FUNCTION_BLOCK TmsHoldStation EXTENDS Process 
VAR
	_EmbarkStation : IStation;
	ExecuteSeqeunce : BOOL;
	HoldMover : I_XtsMover;
	State :(
		Init,                                               
		Ready,                                 
        Waiting,
		Processing,
		Clearing,
		Aborting); 
END_VAR

{analysis -2}

METHOD PUBLIC  Cycle : HRESULT
VAR
	CycleResult : HRESULT;
END_VAR
Cycle := S_OK;
CASE State OF
	Init:
		_Operating := _IsClear := _Complete := _Ready := _HasMover := FALSE;
		StationMovers := 0;
		State := Ready;
	
	Ready:	
		IF ExecuteSeqeunce THEN
			_Operating := _Complete := _HasMover := FALSE;
			_IsClear := _Ready := TRUE;
			StationMovers := 0;
			State := Waiting;
		END_IF
	
	Waiting:
		IF _HasMover THEN
			State := Processing;
			_Operating := TRUE;
			_IsClear := FALSE;
			_Ready := FALSE;
		END_IF
		
	Processing:
		IF _EmbarkStation.IsClear() THEN
			_Complete := TRUE;
			State := Clearing;
		END_IF
		
	Clearing:
		IF NOT _HasMover THEN
			State := Waiting;
			_Operating := FALSE;
			_IsClear := TRUE;
			_Ready := TRUE;
			_Complete := FALSE;
			HoldMover := 0;
		END_IF
		
	Aborting:
		State := Ready;
		HoldMover := 0;
		_HasMover := FALSE;
	ELSE
		Cycle := E_FAIL;
END_CASE
CycleResult := SUPER^.Cycle();

IF CycleResult = E_FAIL THEN
	Cycle := E_FAIL;
END_IF
END_METHOD

METHOD MoverArriving : BOOL
VAR_INPUT
	mover : I_XtsMover;
END_VAR
IF StationMovers <= 2 THEN
	StationMovers := StationMovers + 1;
	HoldMover := mover;
	_HasMover := TRUE;
	MoverArriving := TRUE;
ELSE
	MoverArriving := FALSE;
END_IF
END_METHOD

METHOD PUBLIC MoverAway : BOOL
VAR_INPUT
END_VAR
StationMovers := StationMovers - 1;
IF StationMovers = 0 THEN
	_HasMover := FALSE;
END_IF
HoldMover := 0;
MoverAway := TRUE;
END_METHOD

PROPERTY MyEmbarkStation : IStation
GET
MyEmbarkStation := _EmbarkStation;
END_GET
SET
_EmbarkStation := MyEmbarkStation;
END_SET
END_PROPERTY

METHOD StartStation : BOOL
VAR_INPUT
END_VAR
ExecuteSeqeunce := true;
END_METHOD

METHOD StopStation : BOOL
VAR_INPUT
END_VAR
ExecuteSeqeunce := FALSE;
State := Aborting;
END_METHOD

END_FUNCTION_BLOCK

(* stored: Version 1.1.0.1
   POU TmsHoldStation: Id {f846901d-7486-433e-831a-23bbb539a0bb}, SpecialFunc None
   Method Cycle: Id {c6e1a6e4-2a59-48a3-a2de-6354d31aa549}
   Method MoverArriving: Id {a266c45f-308b-42ff-85d6-9dbbc61ca57d}
   Method MoverAway: Id {1b3a1907-f964-494a-b05a-ec8239679c36}
   Property MyEmbarkStation: Id {32ce3b1d-cc83-40cf-875e-de2f759160d5}
   Get Get: Id {45759e1b-1442-4588-af19-79e9ae38f49e}
   Set Set: Id {51345d54-d899-4179-ae10-0e676d705143}
   Method StartStation: Id {5f526a3c-65d4-46bd-9113-03a24816f81e}
   Method StopStation: Id {0642eca6-8170-4776-8358-60a9a400e4d2} *)
